// TIA Portal V18 export
DATA_BLOCK "FB1523_Weather_Modbus_DB"   // DB8
VERSION : 0.1
// stored: AutoNumber true, DBAccessibleFromOPCUA true, DBAccessibleFromWebserver true, InstanceOfName FB1523_Weather_Modbus, InstanceOfType FB
"FB1523_Weather_Modbus"
   // VAR_INPUT
   //    REQ : Bool;
   //    DISCONNECT : Bool;
   //    ID : CONN_OUC;
   //    IP_1 : Byte;
   //    IP_2 : Byte;
   //    IP_3 : Byte;
   //    IP_4 : Byte;
   //    PORT : UInt;
   // END_VAR
   // VAR_OUTPUT
   //    DONE : Bool;
   //    BUSY : Bool;
   //    ERROR : Bool;
   //    STATUS : Word;
   // END_VAR
   // VAR
   //    CONNECT : TCON_IP_v4;
   //    MB_CLIENT { S7_SetPoint := 'True'} : MB_CLIENT;
   //    RCV_DATA { S7_SetPoint := 'True'} : Array[0..13] of DInt;
   // END_VAR
BEGIN
END_DATA_BLOCK
